// TIA Portal V17 export
// export: Created 2025-08-05T09:35:59.8211144Z, ExportSetting WithDefaults, DisplayName Totally Integrated Automation Portal, DisplayVersion V17, DisplayName TIA Portal Openness, DisplayVersion V17, DisplayName TIA Portal Version Control Interface, DisplayVersion V17, DisplayName SINAMICS Startdrive Advanced, DisplayVersion V17, DisplayName SINAMICS Startdrive G130, G150, S120, S150, SINAMICS MV, S210, DisplayVersion V17, DisplayName SINAMICS Startdrive G110M, G120, G120C, G120D, G120P, G115D, DisplayVersion V17, DisplayName STEP 7 Professional, DisplayVersion V17, DisplayName STEP 7 Safety, DisplayVersion V17, DisplayName WinCC Advanced, DisplayVersion V17
TYPE "typeFaultManagement"
TITLE = Error management / Fehlerverwaltung
// Fehlerverwaltung [V 01.01 | Kernel_V2]
// stored: IsFailsafeCompliant false
   STRUCT
      selectAckFault : Bool;   // Anwahl Störung quittieren (S) / Selection: acknowledge fault (S)
      ackFault : Bool;   // Störung quittieren / Acknowledge fault
      faultGeneral : Bool;   // Generelle Störung steht an / General fault pending
      faultInstantStop : Bool;   // Störung sofort Halt steht an / Fault immediate stop pending
      faultMachineOut : Bool;   // Störung sofort Halt und Maschine Aus steht an / Fault immediate stop and machine off pending
      faultInCycleEnd : Bool;   // Störung Halt nach Taktende steht an / Fault stop at end of cycle pending
      faultNoStop : Bool;   // Störung ohne Stop steht an / Fault without stop pending
      faultActive : Bool;   // Störung ist aktiv (aus eigener oder übergeordeten Gruppen) / Fault is active (from separate or superordinate groups)
      messageGeneral : Bool;   // Meldung steht an / Message pending
      messageOperatorCall : Bool;   // Meldung mit Bedienerruf steht an / Message with operator call pending
      selectInstantStop : Bool;   // Anwahl sofort Halt bei Störung (S) / Selection immediate stop in case of fault (S)
      selectMachineOut : Bool;   // Anwahl sofort Halt und Maschine aus (S)
      selectStopCycleEnd : Bool;   // Anwahl Halt nach Taktende bei Störung (S) / Selection stop at end of cycle in case of fault (S)
      faultInstantStopByParent : Bool;   // Störung sofort Halt von übergeordneter Baugruppe / Fault immediate stop from superordinate assembly
      faultInCycleEndByParent : Bool;   // Störung Halt nach Taktende von übergeordneter Baugruppe / Fault stop at end of cycle from the superordinate assembly
   END_STRUCT;
END_TYPE
